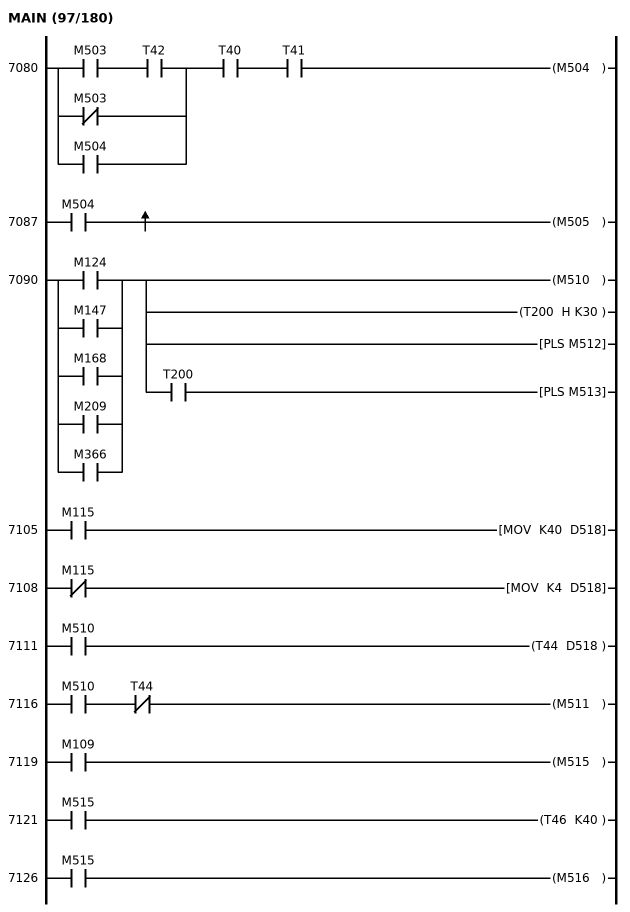
[picture p96: ladder of MAIN, rungs at steps 7080 to 7126]
7080  LD      M503
      AND     T42
      ORI     M503
      OR      M504
      AND     T40
      AND     T41
      OUT     M504
7087  LD      M504
      MEP
      OUT     M505
7090  LD      M124
      OR      M147
      OR      M168
      OR      M209
      OR      M366
      OUT     M510
      OUTH    T200 K30
      PLS     M512
      AND     T200
      PLS     M513
7105  LD      M115
      MOV     K40 D518
7108  LDI     M115
      MOV     K4 D518
7111  LD      M510
      OUT     T44 D518
7116  LD      M510
      ANI     T44
      OUT     M511
7119  LD      M109
      OUT     M515
7121  LD      M515
      OUT     T46 K40
7126  LD      M515
      OUT     M516
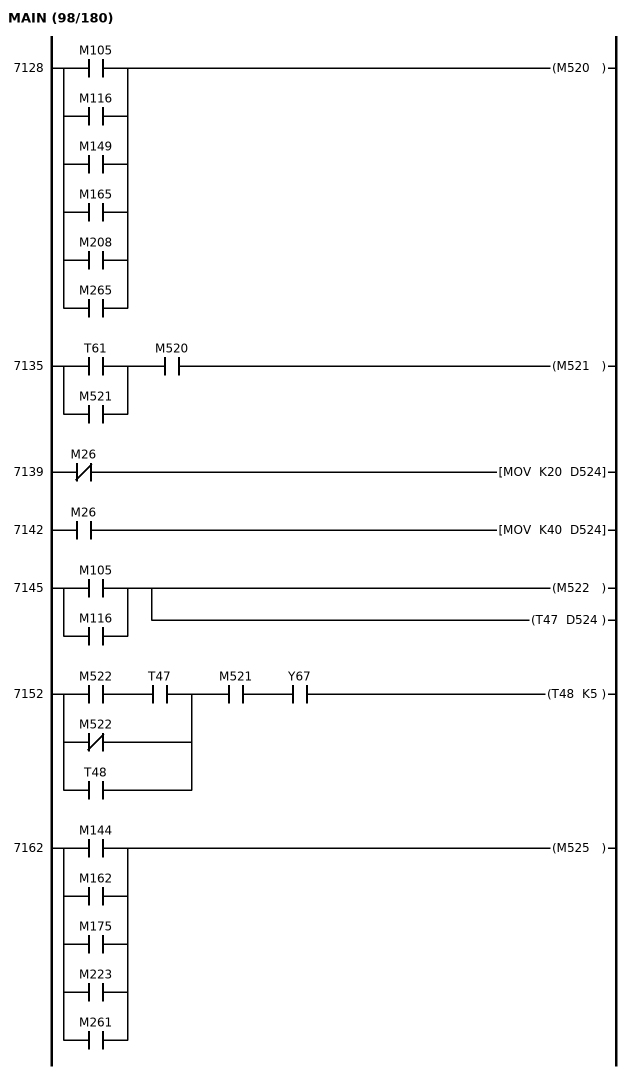
7128  LD      M105
      OR      M116
      OR      M149
      OR      M165
      OR      M208
      OR      M265
      OUT     M520
7135  LD      T61
      OR      M521
      AND     M520
      OUT     M521
7139  LDI     M26
      MOV     K20 D524
7142  LD      M26
      MOV     K40 D524
7145  LD      M105
      OR      M116
      OUT     M522
      OUT     T47 D524
7152  LD      M522
      AND     T47
      ORI     M522
      OR      T48
      AND     M521
      AND     Y67
      OUT     T48 K5
7162  LD      M144
      OR      M162
      OR      M175
      OR      M223
      OR      M261
      OUT     M525
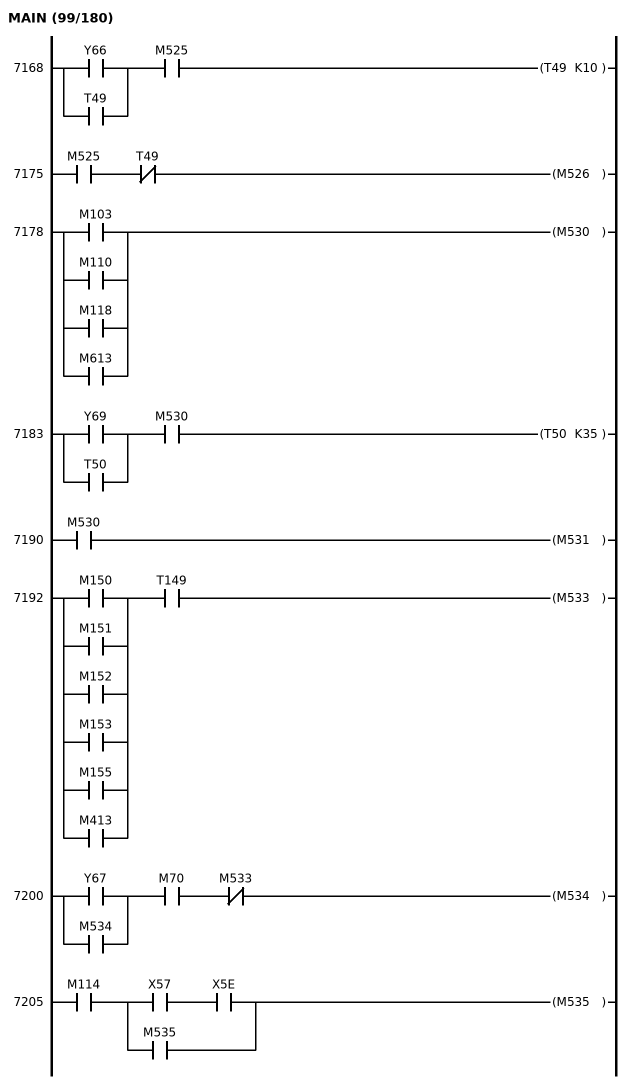
7168  LD      Y66
      OR      T49
      AND     M525
      OUT     T49 K10
7175  LD      M525
      ANI     T49
      OUT     M526
7178  LD      M103
      OR      M110
      OR      M118
      OR      M613
      OUT     M530
7183  LD      Y69
      OR      T50
      AND     M530
      OUT     T50 K35
7190  LD      M530
      OUT     M531
7192  LD      M150
      OR      M151
      OR      M152
      OR      M153
      OR      M155
      OR      M413
      AND     T149
      OUT     M533
7200  LD      Y67
      OR      M534
      AND     M70
      ANI     M533
      OUT     M534
7205  LD      M114
      LD      X57
      AND     X5E
      OR      M535
      ANB
      OUT     M535
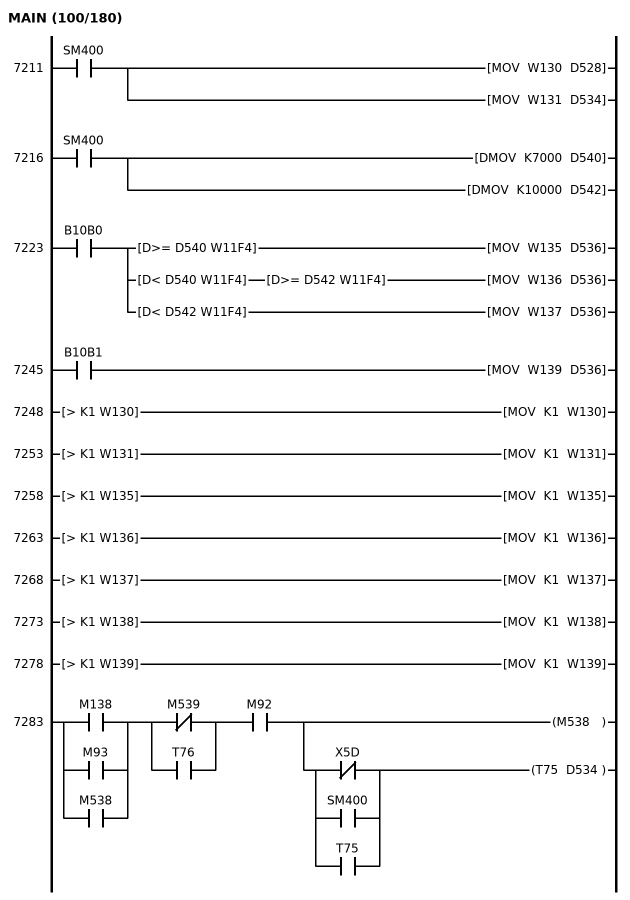
7211  LD      SM400
      MOV     W130 D528
      MOV     W131 D534
7216  LD      SM400
      DMOV    K7000 D540
      DMOV    K10000 D542
7223  LD      B10B0
      MPS
      ANDD>=  D540 W11F4
      MOV     W135 D536
      MRD
      ANDD<   D540 W11F4
      ANDD>=  D542 W11F4
      MOV     W136 D536
      MPP
      ANDD<   D542 W11F4
      MOV     W137 D536
7245  LD      B10B1
      MOV     W139 D536
7248  LD>     K1 W130
      MOV     K1 W130
7253  LD>     K1 W131
      MOV     K1 W131
7258  LD>     K1 W135
      MOV     K1 W135
7263  LD>     K1 W136
      MOV     K1 W136
7268  LD>     K1 W137
      MOV     K1 W137
7273  LD>     K1 W138
      MOV     K1 W138
7278  LD>     K1 W139
      MOV     K1 W139
7283  LD      M138
      OR      M93
      OR      M538
      LDI     M539
      OR      T76
      ANB
      AND     M92
      OUT     M538
      LDI     X5D
      OR      SM400
      OR      T75
      ANB
      OUT     T75 D534
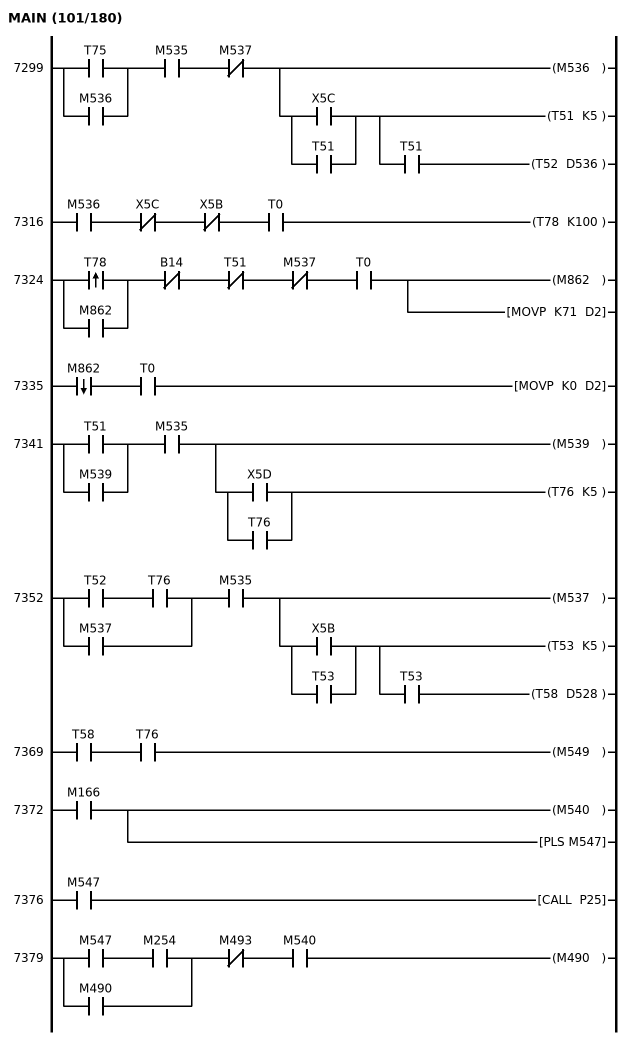
7299  LD      T75
      OR      M536
      AND     M535
      ANI     M537
      OUT     M536
      LD      X5C
      OR      T51
      ANB
      OUT     T51 K5
      AND     T51
      OUT     T52 D536
7316  LD      M536
      ANI     X5C
      ANI     X5B
      AND     T0
      OUT     T78 K100
7324  LDP     T78
      OR      M862
      ANI     B14
      ANI     T51
      ANI     M537
      AND     T0
      OUT     M862
      MOVP    K71 D2
7335  LDF     M862
      AND     T0
      MOVP    K0 D2
7341  LD      T51
      OR      M539
      AND     M535
      OUT     M539
      LD      X5D
      OR      T76
      ANB
      OUT     T76 K5
7352  LD      T52
      AND     T76
      OR      M537
      AND     M535
      OUT     M537
      LD      X5B
      OR      T53
      ANB
      OUT     T53 K5
      AND     T53
      OUT     T58 D528
7369  LD      T58
      AND     T76
      OUT     M549
7372  LD      M166
      OUT     M540
      PLS     M547
7376  LD      M547
      CALL    P25
7379  LD      M547
      AND     M254
      OR      M490
      ANI     M493
      AND     M540
      OUT     M490
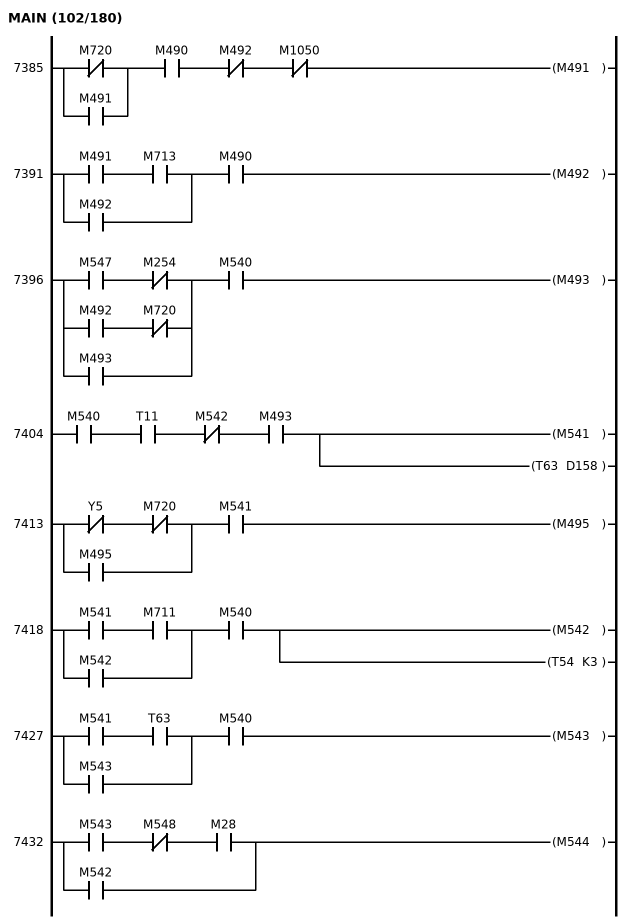
7385  LDI     M720
      OR      M491
      AND     M490
      ANI     M492
      ANI     M1050
      OUT     M491
7391  LD      M491
      AND     M713
      OR      M492
      AND     M490
      OUT     M492
7396  LD      M547
      ANI     M254
      LD      M492
      ANI     M720
      ORB
      OR      M493
      AND     M540
      OUT     M493
7404  LD      M540
      AND     T11
      ANI     M542
      AND     M493
      OUT     M541
      OUT     T63 D158
7413  LDI     Y5
      ANI     M720
      OR      M495
      AND     M541
      OUT     M495
7418  LD      M541
      AND     M711
      OR      M542
      AND     M540
      OUT     M542
      OUT     T54 K3
7427  LD      M541
      AND     T63
      OR      M543
      AND     M540
      OUT     M543
7432  LD      M543
      ANI     M548
      AND     M28
      OR      M542
      OUT     M544
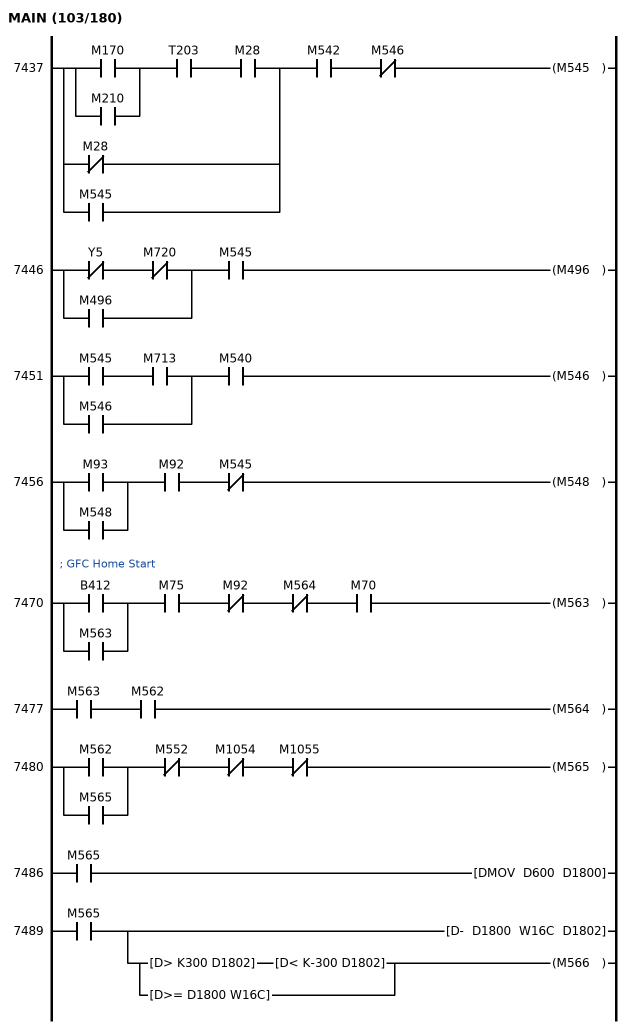
7437  LD      M170
      OR      M210
      AND     T203
      AND     M28
      ORI     M28
      OR      M545
      AND     M542
      ANI     M546
      OUT     M545
7446  LDI     Y5
      ANI     M720
      OR      M496
      AND     M545
      OUT     M496
7451  LD      M545
      AND     M713
      OR      M546
      AND     M540
      OUT     M546
7456  LD      M93
      OR      M548
      AND     M92
      ANI     M545
      OUT     M548
; GFC Home Start
7470  LD      B412
      OR      M563
      AND     M75
      ANI     M92
      ANI     M564
      AND     M70
      OUT     M563
7477  LD      M563
      AND     M562
      OUT     M564
7480  LD      M562
      OR      M565
      ANI     M552
      ANI     M1054
      ANI     M1055
      OUT     M565
7486  LD      M565
      DMOV    D600 D1800
7489  LD      M565
      D-      D1800 W16C D1802
      LDD>    K300 D1802
      ANDD<   K-300 D1802
      ORD>=   D1800 W16C
      ANB
      OUT     M566
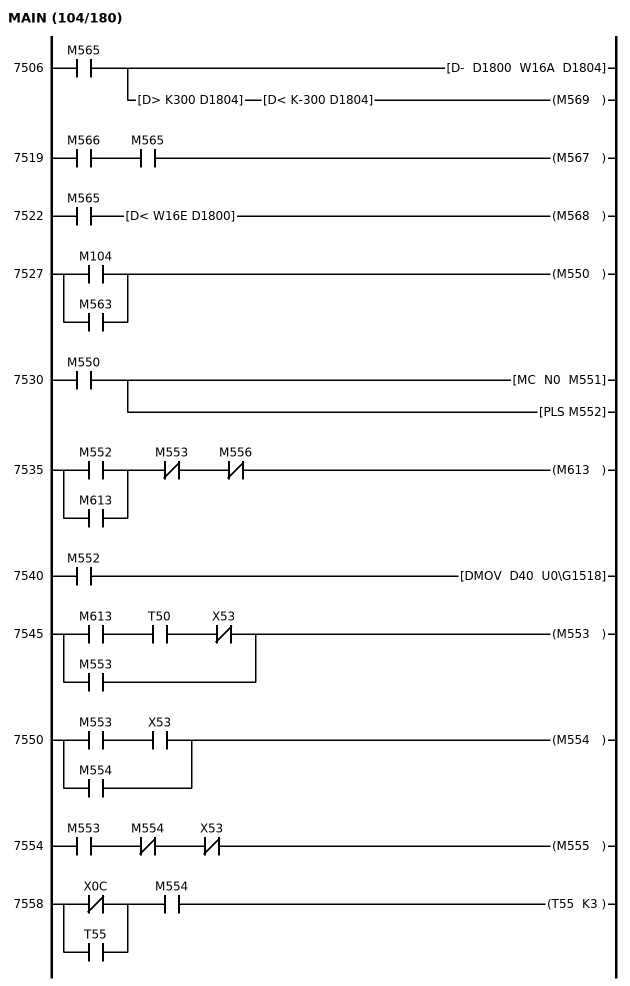
7506  LD      M565
      D-      D1800 W16A D1804
      ANDD>   K300 D1804
      ANDD<   K-300 D1804
      OUT     M569
7519  LD      M566
      AND     M565
      OUT     M567
7522  LD      M565
      ANDD<   W16E D1800
      OUT     M568
7527  LD      M104
      OR      M563
      OUT     M550
7530  LD      M550
      MC      N0 M551
      PLS     M552
7535  LD      M552
      OR      M613
      ANI     M553
      ANI     M556
      OUT     M613
7540  LD      M552
      DMOV    D40 U0\G1518
7545  LD      M613
      AND     T50
      ANI     X53
      OR      M553
      OUT     M553
7550  LD      M553
      AND     X53
      OR      M554
      OUT     M554
7554  LD      M553
      ANI     M554
      ANI     X53
      OUT     M555
7558  LDI     X0C
      OR      T55
      AND     M554
      OUT     T55 K3
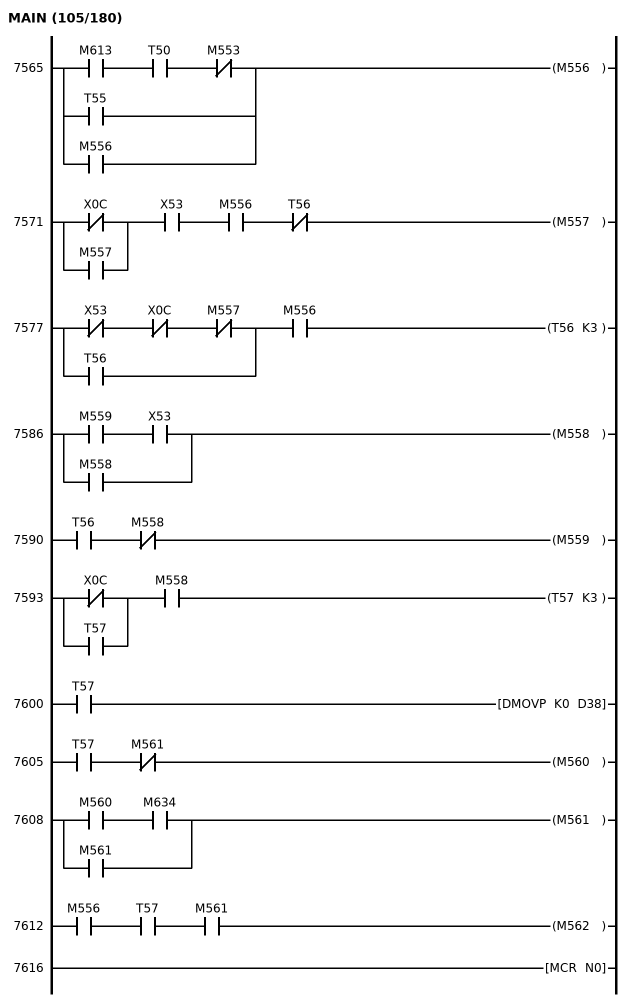
7565  LD      M613
      AND     T50
      ANI     M553
      OR      T55
      OR      M556
      OUT     M556
7571  LDI     X0C
      OR      M557
      AND     X53
      AND     M556
      ANI     T56
      OUT     M557
7577  LDI     X53
      ANI     X0C
      ANI     M557
      OR      T56
      AND     M556
      OUT     T56 K3
7586  LD      M559
      AND     X53
      OR      M558
      OUT     M558
7590  LD      T56
      ANI     M558
      OUT     M559
7593  LDI     X0C
      OR      T57
      AND     M558
      OUT     T57 K3
7600  LD      T57
      DMOVP   K0 D38
7605  LD      T57
      ANI     M561
      OUT     M560
7608  LD      M560
      AND     M634
      OR      M561
      OUT     M561
7612  LD      M556
      AND     T57
      AND     M561
      OUT     M562
7616  MCR     N0
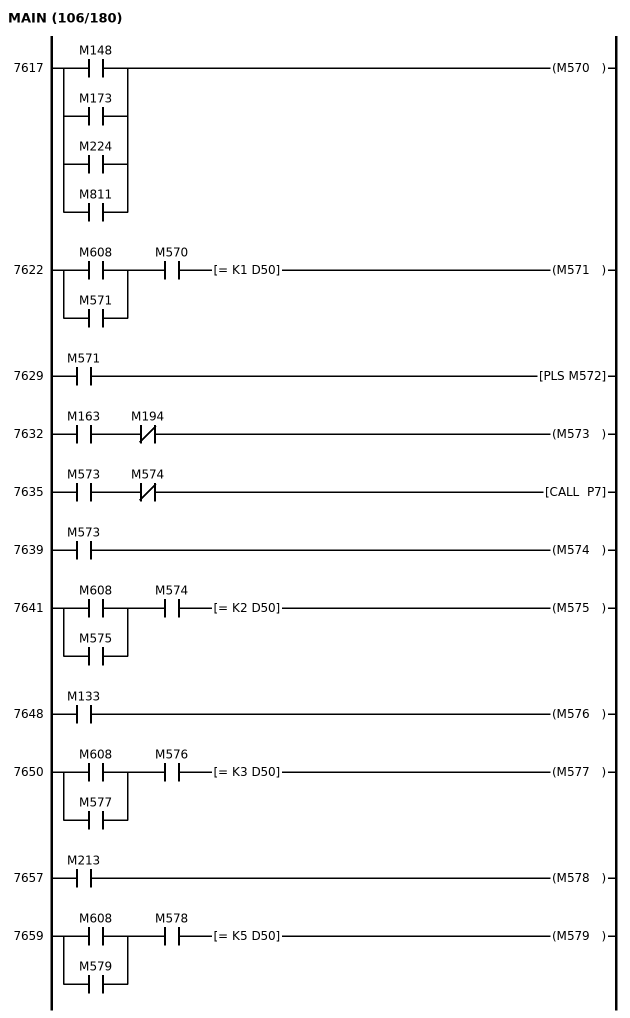
7617  LD      M148
      OR      M173
      OR      M224
      OR      M811
      OUT     M570
7622  LD      M608
      OR      M571
      AND     M570
      AND=    K1 D50
      OUT     M571
7629  LD      M571
      PLS     M572
7632  LD      M163
      ANI     M194
      OUT     M573
7635  LD      M573
      ANI     M574
      CALL    P7
7639  LD      M573
      OUT     M574
7641  LD      M608
      OR      M575
      AND     M574
      AND=    K2 D50
      OUT     M575
7648  LD      M133
      OUT     M576
7650  LD      M608
      OR      M577
      AND     M576
      AND=    K3 D50
      OUT     M577
7657  LD      M213
      OUT     M578
7659  LD      M608
      OR      M579
      AND     M578
      AND=    K5 D50
      OUT     M579
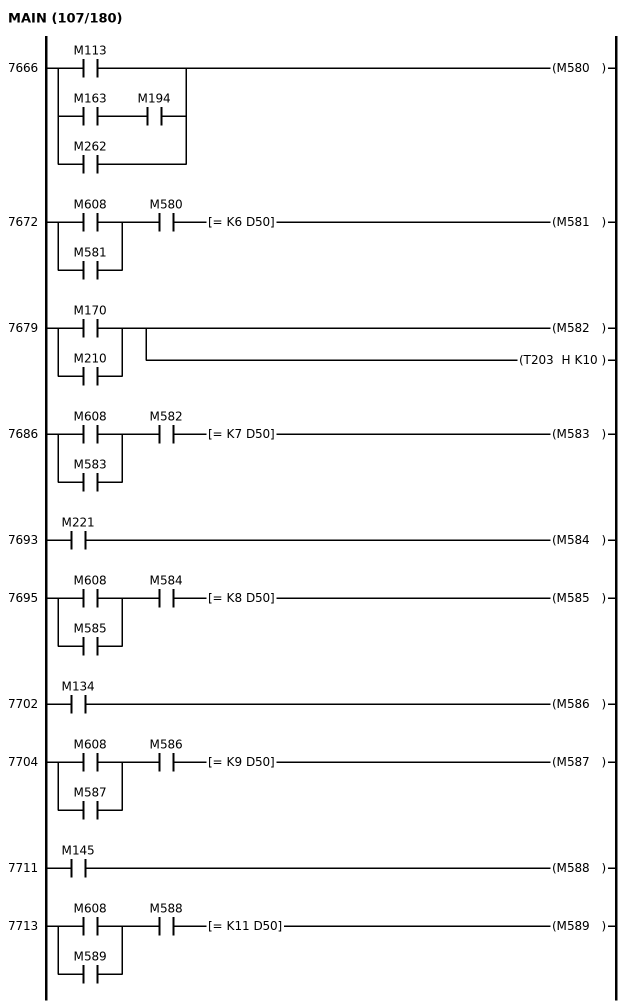
7666  LD      M113
      LD      M163
      AND     M194
      ORB
      OR      M262
      OUT     M580
7672  LD      M608
      OR      M581
      AND     M580
      AND=    K6 D50
      OUT     M581
7679  LD      M170
      OR      M210
      OUT     M582
      OUTH    T203 K10
7686  LD      M608
      OR      M583
      AND     M582
      AND=    K7 D50
      OUT     M583
7693  LD      M221
      OUT     M584
7695  LD      M608
      OR      M585
      AND     M584
      AND=    K8 D50
      OUT     M585
7702  LD      M134
      OUT     M586
7704  LD      M608
      OR      M587
      AND     M586
      AND=    K9 D50
      OUT     M587
7711  LD      M145
      OUT     M588
7713  LD      M608
      OR      M589
      AND     M588
      AND=    K11 D50
      OUT     M589
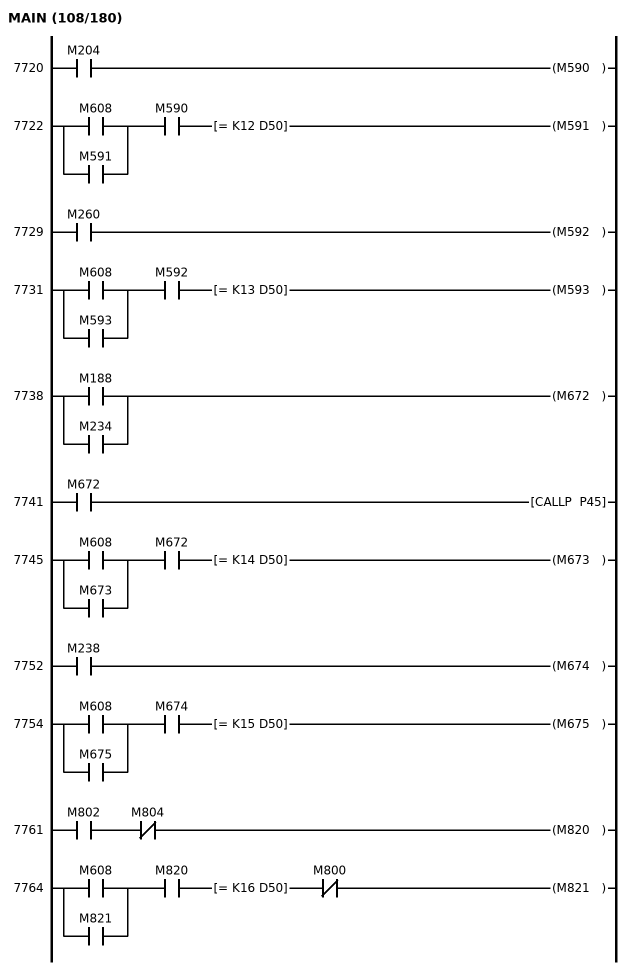
7720  LD      M204
      OUT     M590
7722  LD      M608
      OR      M591
      AND     M590
      AND=    K12 D50
      OUT     M591
7729  LD      M260
      OUT     M592
7731  LD      M608
      OR      M593
      AND     M592
      AND=    K13 D50
      OUT     M593
7738  LD      M188
      OR      M234
      OUT     M672
7741  LD      M672
      CALLP   P45
7745  LD      M608
      OR      M673
      AND     M672
      AND=    K14 D50
      OUT     M673
7752  LD      M238
      OUT     M674
7754  LD      M608
      OR      M675
      AND     M674
      AND=    K15 D50
      OUT     M675
7761  LD      M802
      ANI     M804
      OUT     M820
7764  LD      M608
      OR      M821
      AND     M820
      AND=    K16 D50
      ANI     M800
      OUT     M821
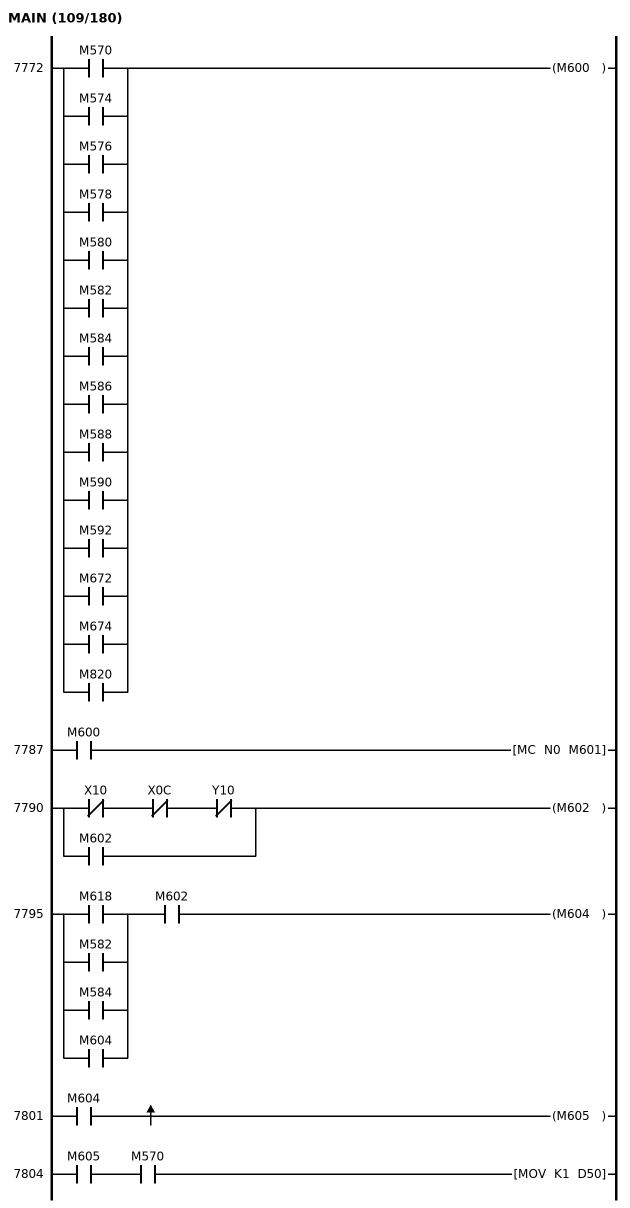
7772  LD      M570
      OR      M574
      OR      M576
      OR      M578
      OR      M580
      OR      M582
      OR      M584
      OR      M586
      OR      M588
      OR      M590
      OR      M592
      OR      M672
      OR      M674
      OR      M820
      OUT     M600
7787  LD      M600
      MC      N0 M601
7790  LDI     X10
      ANI     X0C
      ANI     Y10
      OR      M602
      OUT     M602
7795  LD      M618
      OR      M582
      OR      M584
      OR      M604
      AND     M602
      OUT     M604
7801  LD      M604
      MEP
      OUT     M605
7804  LD      M605
      AND     M570
      MOV     K1 D50
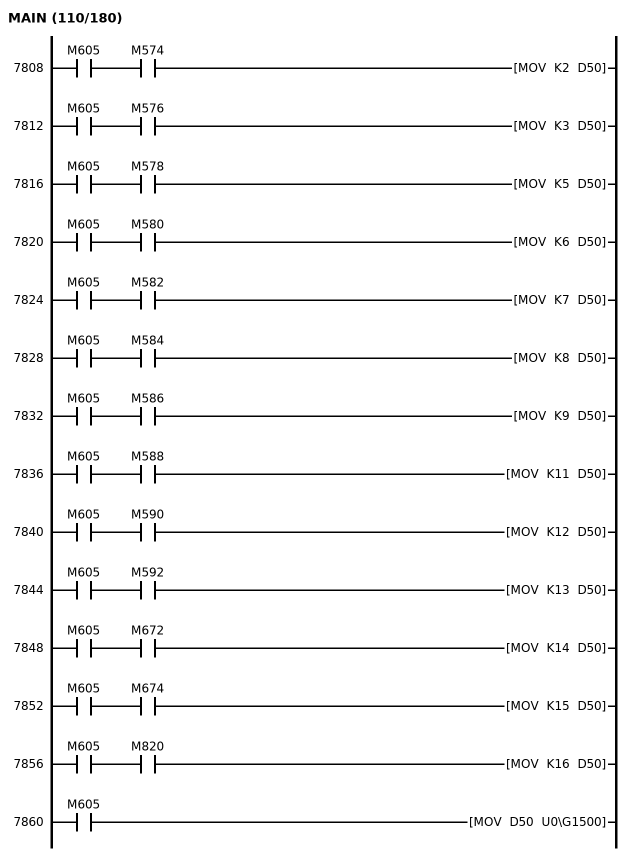
7808  LD      M605
      AND     M574
      MOV     K2 D50
7812  LD      M605
      AND     M576
      MOV     K3 D50
7816  LD      M605
      AND     M578
      MOV     K5 D50
7820  LD      M605
      AND     M580
      MOV     K6 D50
7824  LD      M605
      AND     M582
      MOV     K7 D50
7828  LD      M605
      AND     M584
      MOV     K8 D50
7832  LD      M605
      AND     M586
      MOV     K9 D50
7836  LD      M605
      AND     M588
      MOV     K11 D50
7840  LD      M605
      AND     M590
      MOV     K12 D50
7844  LD      M605
      AND     M592
      MOV     K13 D50
7848  LD      M605
      AND     M672
      MOV     K14 D50
7852  LD      M605
      AND     M674
      MOV     K15 D50
7856  LD      M605
      AND     M820
      MOV     K16 D50
7860  LD      M605
      MOV     D50 U0\G1500
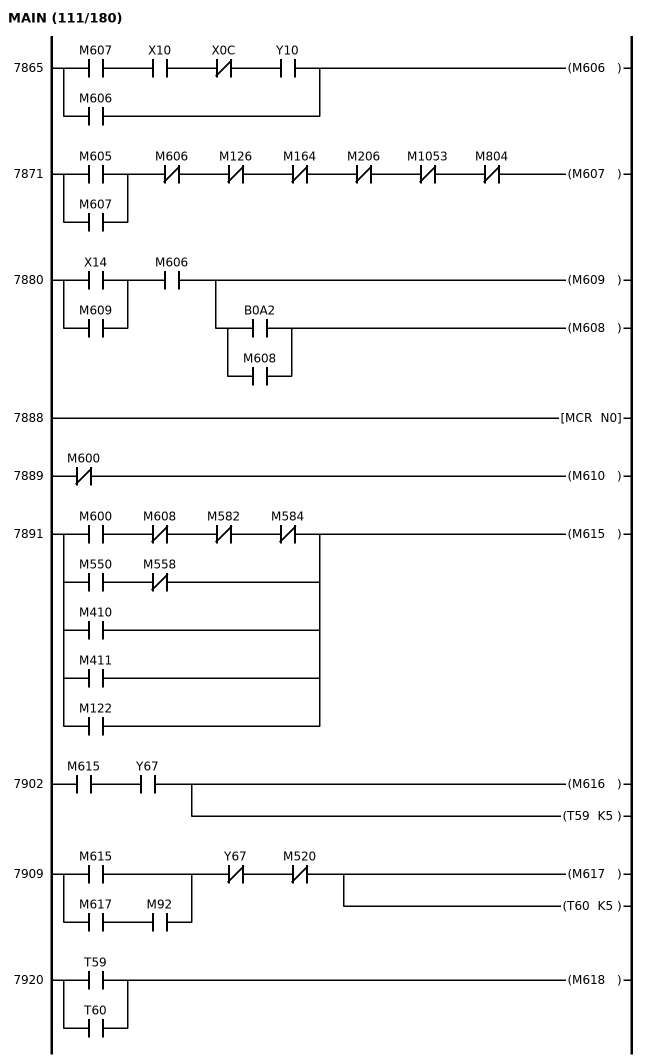
7865  LD      M607
      AND     X10
      ANI     X0C
      AND     Y10
      OR      M606
      OUT     M606
7871  LD      M605
      OR      M607
      ANI     M606
      ANI     M126
      ANI     M164
      ANI     M206
      ANI     M1053
      ANI     M804
      OUT     M607
7880  LD      X14
      OR      M609
      AND     M606
      OUT     M609
      LD      B0A2
      OR      M608
      ANB
      OUT     M608
7888  MCR     N0
7889  LDI     M600
      OUT     M610
7891  LD      M600
      ANI     M608
      ANI     M582
      ANI     M584
      LD      M550
      ANI     M558
      ORB
      OR      M410
      OR      M411
      OR      M122
      OUT     M615
7902  LD      M615
      AND     Y67
      OUT     M616
      OUT     T59 K5
7909  LD      M615
      LD      M617
      AND     M92
      ORB
      ANI     Y67
      ANI     M520
      OUT     M617
      OUT     T60 K5
7920  LD      T59
      OR      T60
      OUT     M618
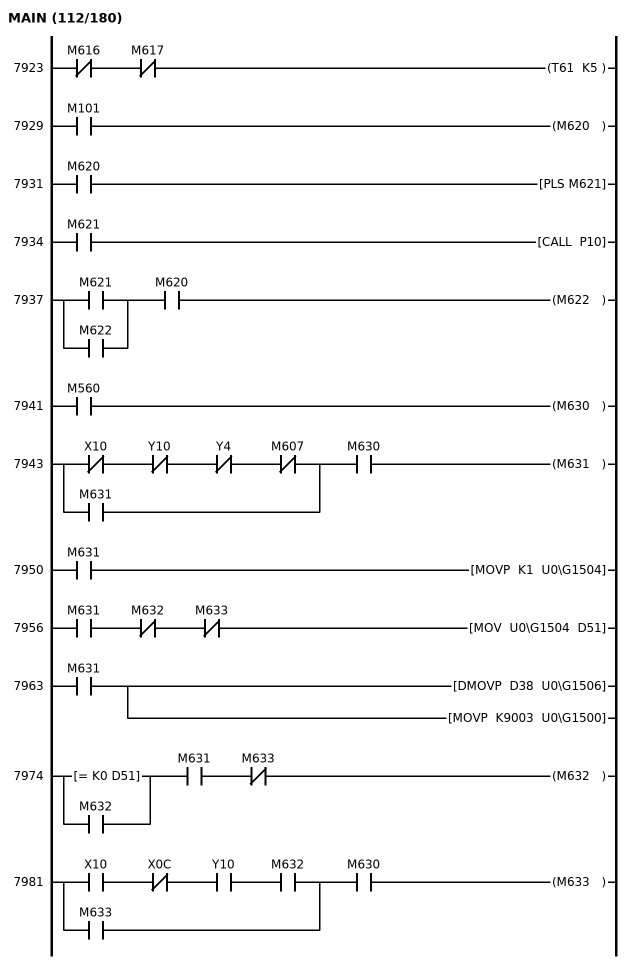
7923  LDI     M616
      ANI     M617
      OUT     T61 K5
7929  LD      M101
      OUT     M620
7931  LD      M620
      PLS     M621
7934  LD      M621
      CALL    P10
7937  LD      M621
      OR      M622
      AND     M620
      OUT     M622
7941  LD      M560
      OUT     M630
7943  LDI     X10
      ANI     Y10
      ANI     Y4
      ANI     M607
      OR      M631
      AND     M630
      OUT     M631
7950  LD      M631
      MOVP    K1 U0\G1504
7956  LD      M631
      ANI     M632
      ANI     M633
      MOV     U0\G1504 D51
7963  LD      M631
      DMOVP   D38 U0\G1506
      MOVP    K9003 U0\G1500
7974  LD=     K0 D51
      OR      M632
      AND     M631
      ANI     M633
      OUT     M632
7981  LD      X10
      ANI     X0C
      AND     Y10
      AND     M632
      OR      M633
      AND     M630
      OUT     M633
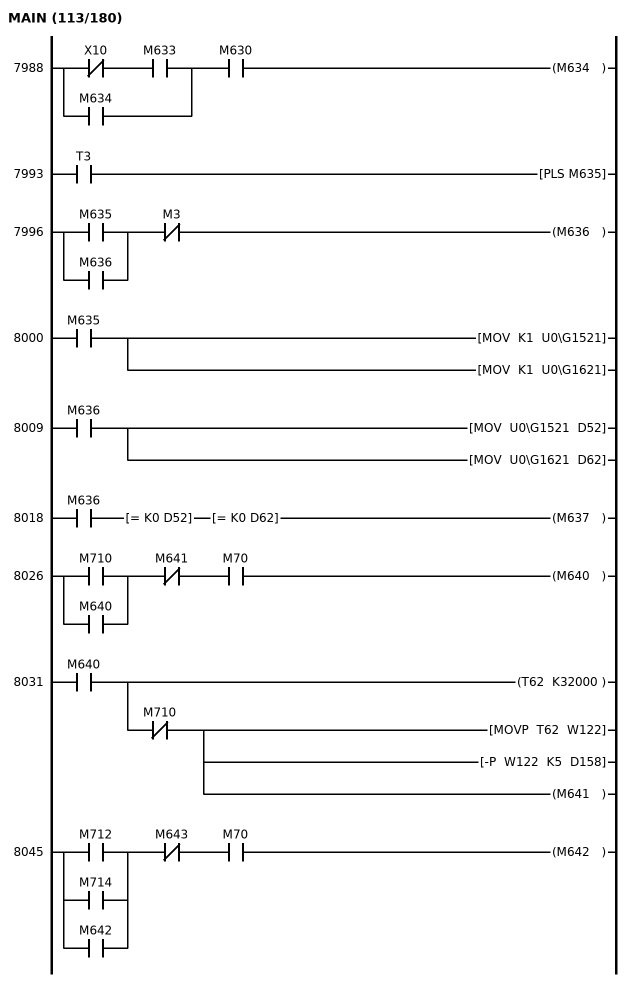
7988  LDI     X10
      AND     M633
      OR      M634
      AND     M630
      OUT     M634
7993  LD      T3
      PLS     M635
7996  LD      M635
      OR      M636
      ANI     M3
      OUT     M636
8000  LD      M635
      MOV     K1 U0\G1521
      MOV     K1 U0\G1621
8009  LD      M636
      MOV     U0\G1521 D52
      MOV     U0\G1621 D62
8018  LD      M636
      AND=    K0 D52
      AND=    K0 D62
      OUT     M637
8026  LD      M710
      OR      M640
      ANI     M641
      AND     M70
      OUT     M640
8031  LD      M640
      OUT     T62 K32000
      ANI     M710
      MOVP    T62 W122
      -P      W122 K5 D158
      OUT     M641
8045  LD      M712
      OR      M714
      OR      M642
      ANI     M643
      AND     M70
      OUT     M642
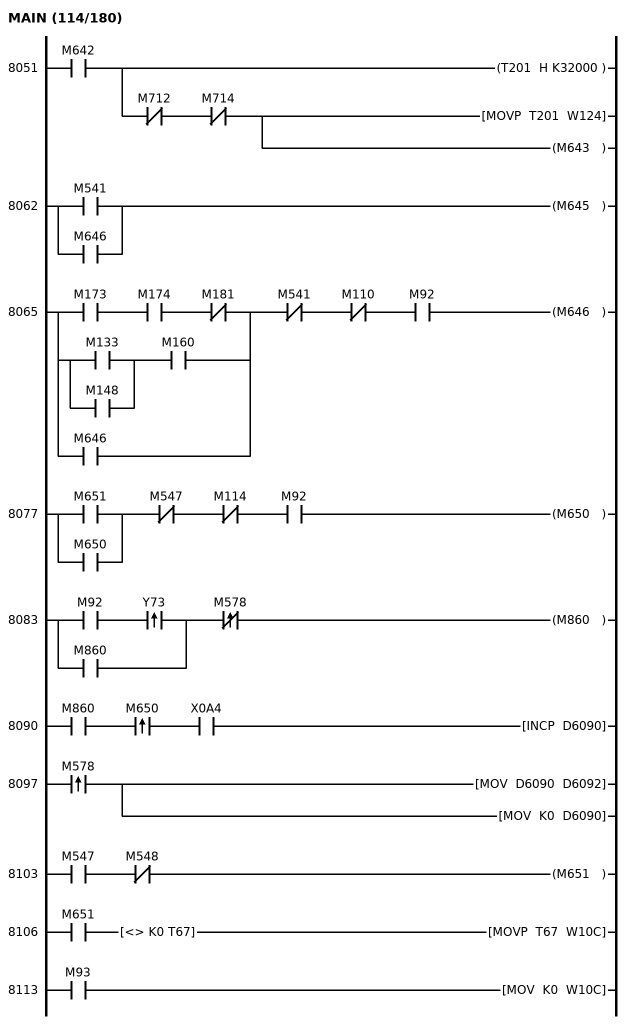
8051  LD      M642
      OUTH    T201 K32000
      ANI     M712
      ANI     M714
      MOVP    T201 W124
      OUT     M643
8062  LD      M541
      OR      M646
      OUT     M645
8065  LD      M173
      AND     M174
      ANI     M181
      LD      M133
      OR      M148
      AND     M160
      ORB
      OR      M646
      ANI     M541
      ANI     M110
      AND     M92
      OUT     M646
8077  LD      M651
      OR      M650
      ANI     M547
      ANI     M114
      AND     M92
      OUT     M650
8083  LD      M92
      ANDP    Y73
      OR      M860
      ANDPI   M578
      OUT     M860
8090  LD      M860
      ANDP    M650
      AND     X0A4
      INCP    D6090
8097  LDP     M578
      MOV     D6090 D6092
      MOV     K0 D6090
8103  LD      M547
      ANI     M548
      OUT     M651
8106  LD      M651
      AND<>   K0 T67
      MOVP    T67 W10C
8113  LD      M93
      MOV     K0 W10C
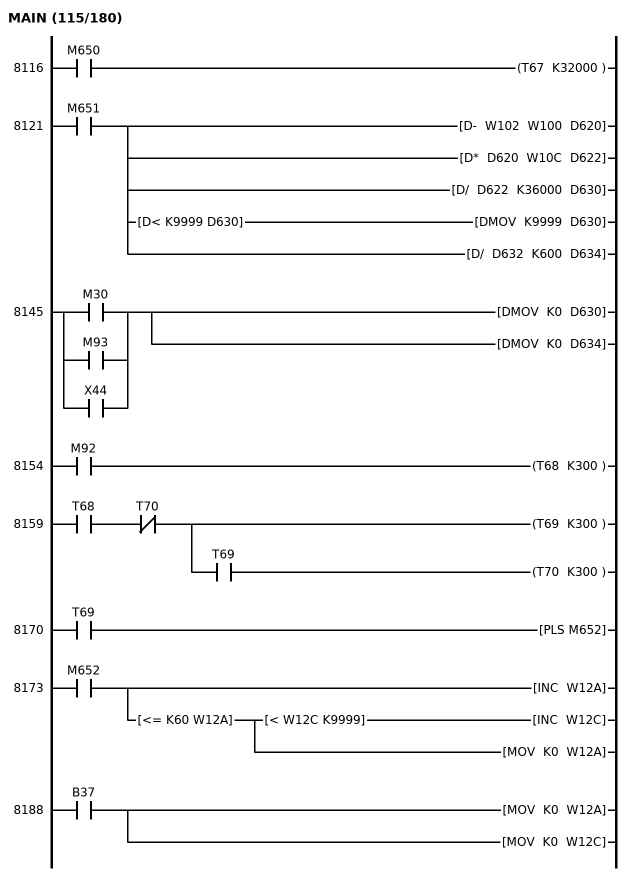
8116  LD      M650
      OUT     T67 K32000
8121  LD      M651
      D-      W102 W100 D620
      D*      D620 W10C D622
      D/      D622 K36000 D630
      MPS
      ANDD<   K9999 D630
      DMOV    K9999 D630
      MPP
      D/      D632 K600 D634
8145  LD      M30
      OR      M93
      OR      X44
      DMOV    K0 D630
      DMOV    K0 D634
8154  LD      M92
      OUT     T68 K300
8159  LD      T68
      ANI     T70
      OUT     T69 K300
      AND     T69
      OUT     T70 K300
8170  LD      T69
      PLS     M652
8173  LD      M652
      INC     W12A
      AND<=   K60 W12A
      MPS
      AND<    W12C K9999
      INC     W12C
      MPP
      MOV     K0 W12A
8188  LD      B37
      MOV     K0 W12A
      MOV     K0 W12C
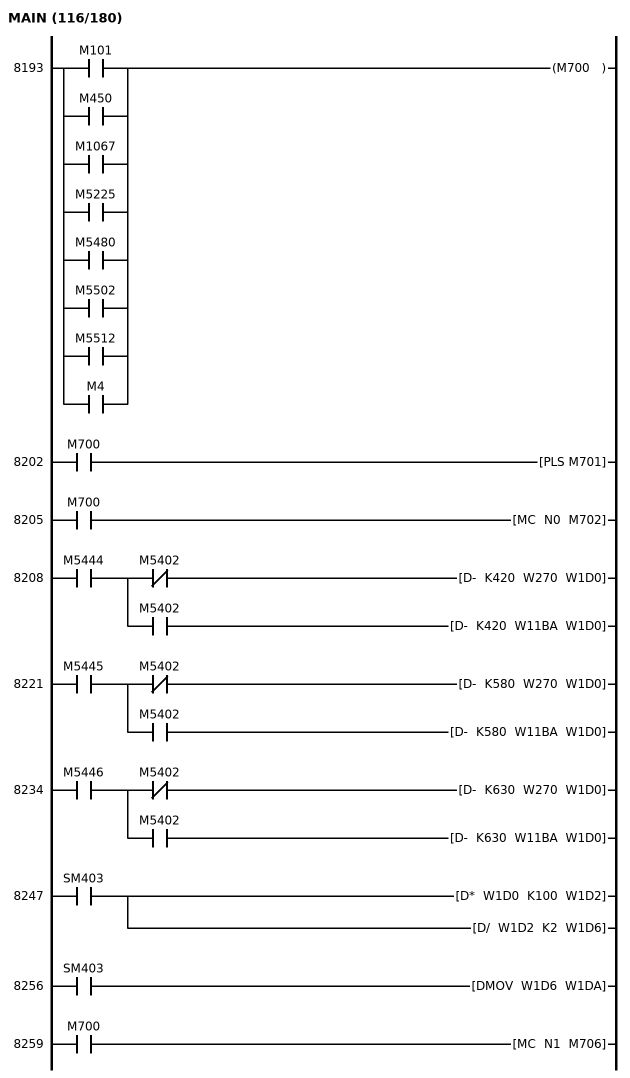
8193  LD      M101
      OR      M450
      OR      M1067
      OR      M5225
      OR      M5480
      OR      M5502
      OR      M5512
      OR      M4
      OUT     M700
8202  LD      M700
      PLS     M701
8205  LD      M700
      MC      N0 M702
8208  LD      M5444
      MPS
      ANI     M5402
      D-      K420 W270 W1D0
      MPP
      AND     M5402
      D-      K420 W11BA W1D0
8221  LD      M5445
      MPS
      ANI     M5402
      D-      K580 W270 W1D0
      MPP
      AND     M5402
      D-      K580 W11BA W1D0
8234  LD      M5446
      MPS
      ANI     M5402
      D-      K630 W270 W1D0
      MPP
      AND     M5402
      D-      K630 W11BA W1D0
8247  LD      SM403
      D*      W1D0 K100 W1D2
      D/      W1D2 K2 W1D6
8256  LD      SM403
      DMOV    W1D6 W1DA
8259  LD      M700
      MC      N1 M706
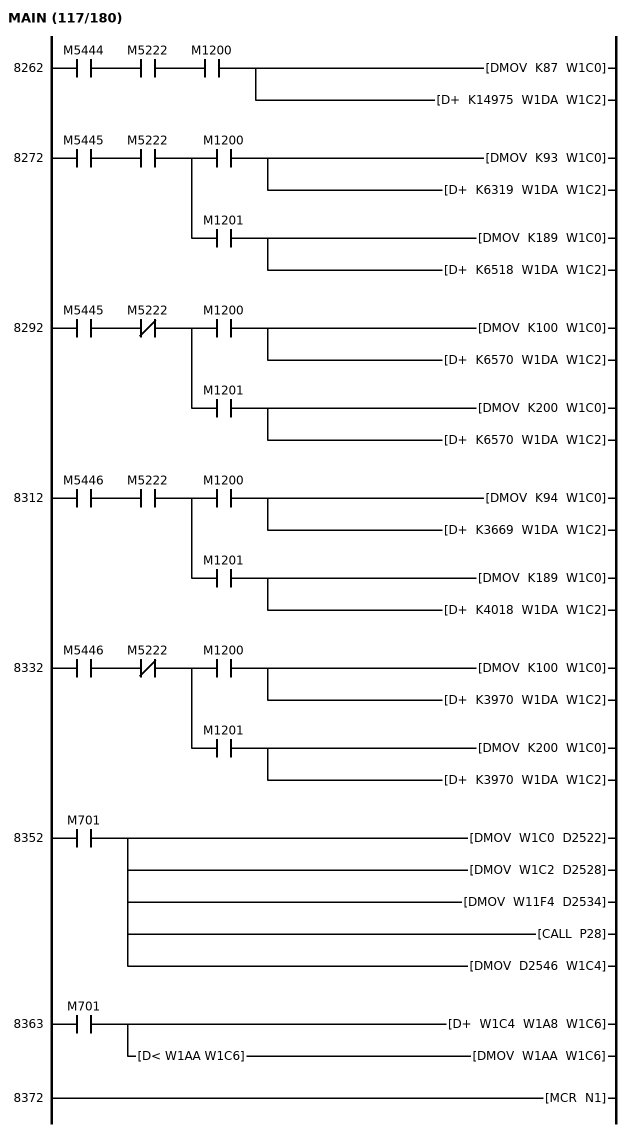
8262  LD      M5444
      AND     M5222
      AND     M1200
      DMOV    K87 W1C0
      D+      K14975 W1DA W1C2
8272  LD      M5445
      AND     M5222
      MPS
      AND     M1200
      DMOV    K93 W1C0
      D+      K6319 W1DA W1C2
      MPP
      AND     M1201
      DMOV    K189 W1C0
      D+      K6518 W1DA W1C2
8292  LD      M5445
      ANI     M5222
      MPS
      AND     M1200
      DMOV    K100 W1C0
      D+      K6570 W1DA W1C2
      MPP
      AND     M1201
      DMOV    K200 W1C0
      D+      K6570 W1DA W1C2
8312  LD      M5446
      AND     M5222
      MPS
      AND     M1200
      DMOV    K94 W1C0
      D+      K3669 W1DA W1C2
      MPP
      AND     M1201
      DMOV    K189 W1C0
      D+      K4018 W1DA W1C2
8332  LD      M5446
      ANI     M5222
      MPS
      AND     M1200
      DMOV    K100 W1C0
      D+      K3970 W1DA W1C2
      MPP
      AND     M1201
      DMOV    K200 W1C0
      D+      K3970 W1DA W1C2
8352  LD      M701
      DMOV    W1C0 D2522
      DMOV    W1C2 D2528
      DMOV    W11F4 D2534
      CALL    P28
      DMOV    D2546 W1C4
8363  LD      M701
      D+      W1C4 W1A8 W1C6
      ANDD<   W1AA W1C6
      DMOV    W1AA W1C6
8372  MCR     N1
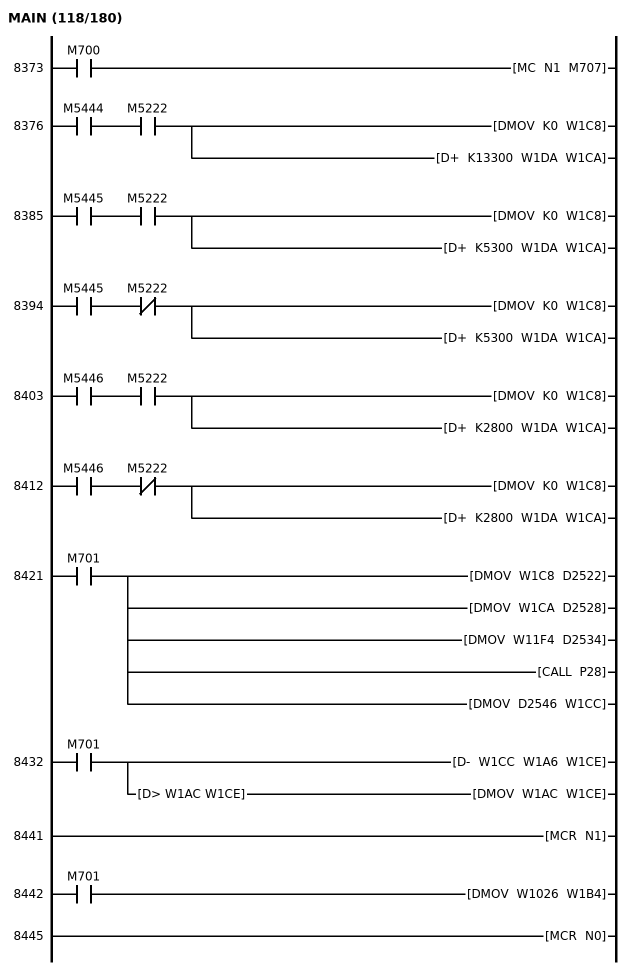
8373  LD      M700
      MC      N1 M707
8376  LD      M5444
      AND     M5222
      DMOV    K0 W1C8
      D+      K13300 W1DA W1CA
8385  LD      M5445
      AND     M5222
      DMOV    K0 W1C8
      D+      K5300 W1DA W1CA
8394  LD      M5445
      ANI     M5222
      DMOV    K0 W1C8
      D+      K5300 W1DA W1CA
8403  LD      M5446
      AND     M5222
      DMOV    K0 W1C8
      D+      K2800 W1DA W1CA
8412  LD      M5446
      ANI     M5222
      DMOV    K0 W1C8
      D+      K2800 W1DA W1CA
8421  LD      M701
      DMOV    W1C8 D2522
      DMOV    W1CA D2528
      DMOV    W11F4 D2534
      CALL    P28
      DMOV    D2546 W1CC
8432  LD      M701
      D-      W1CC W1A6 W1CE
      ANDD>   W1AC W1CE
      DMOV    W1AC W1CE
8441  MCR     N1
8442  LD      M701
      DMOV    W1026 W1B4
8445  MCR     N0
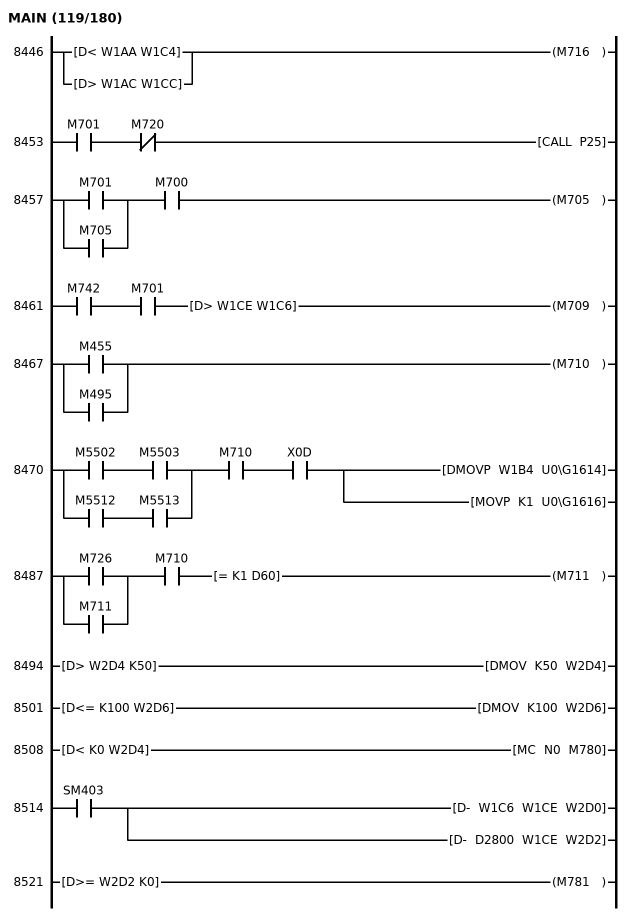
8446  LDD<    W1AA W1C4
      ORD>    W1AC W1CC
      OUT     M716
8453  LD      M701
      ANI     M720
      CALL    P25
8457  LD      M701
      OR      M705
      AND     M700
      OUT     M705
8461  LD      M742
      AND     M701
      ANDD>   W1CE W1C6
      OUT     M709
8467  LD      M455
      OR      M495
      OUT     M710
8470  LD      M5502
      AND     M5503
      LD      M5512
      AND     M5513
      ORB
      AND     M710
      AND     X0D
      DMOVP   W1B4 U0\G1614
      MOVP    K1 U0\G1616
8487  LD      M726
      OR      M711
      AND     M710
      AND=    K1 D60
      OUT     M711
8494  LDD>    W2D4 K50
      DMOV    K50 W2D4
8501  LDD<=   K100 W2D6
      DMOV    K100 W2D6
8508  LDD<    K0 W2D4
      MC      N0 M780
8514  LD      SM403
      D-      W1C6 W1CE W2D0
      D-      D2800 W1CE W2D2
8521  LDD>=   W2D2 K0
      OUT     M781
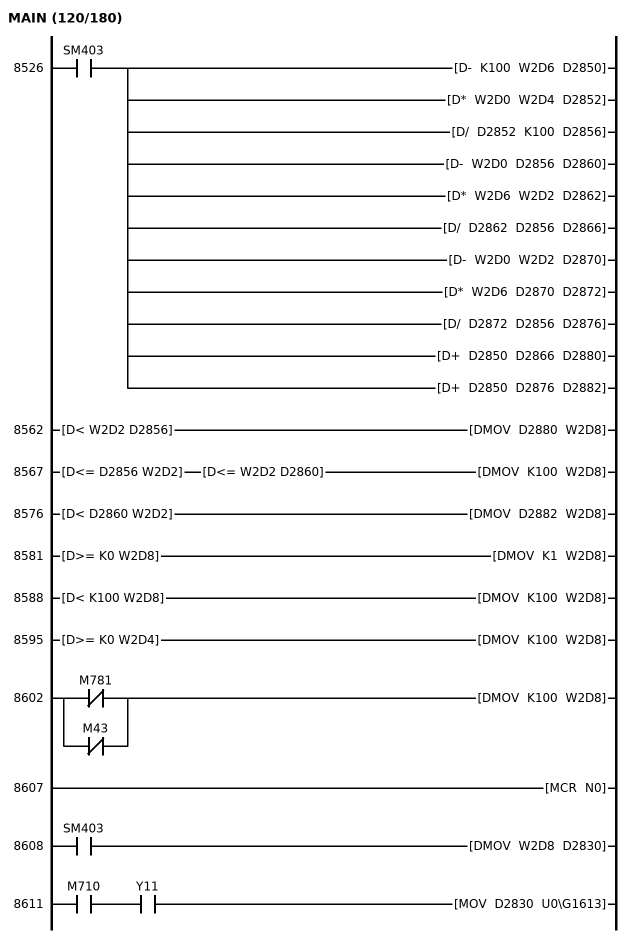
8526  LD      SM403
      D-      K100 W2D6 D2850
      D*      W2D0 W2D4 D2852
      D/      D2852 K100 D2856
      D-      W2D0 D2856 D2860
      D*      W2D6 W2D2 D2862
      D/      D2862 D2856 D2866
      D-      W2D0 W2D2 D2870
      D*      W2D6 D2870 D2872
      D/      D2872 D2856 D2876
      D+      D2850 D2866 D2880
      D+      D2850 D2876 D2882
8562  LDD<    W2D2 D2856
      DMOV    D2880 W2D8
8567  LDD<=   D2856 W2D2
      ANDD<=  W2D2 D2860
      DMOV    K100 W2D8
8576  LDD<    D2860 W2D2
      DMOV    D2882 W2D8
8581  LDD>=   K0 W2D8
      DMOV    K1 W2D8
8588  LDD<    K100 W2D8
      DMOV    K100 W2D8
8595  LDD>=   K0 W2D4
      DMOV    K100 W2D8
8602  LDI     M781
      ORI     M43
      DMOV    K100 W2D8
8607  MCR     N0
8608  LD      SM403
      DMOV    W2D8 D2830
8611  LD      M710
      AND     Y11
      MOV     D2830 U0\G1613
